(* PLC project Unnamed, Unknown Unnamed 1 *)
(* stored: creationDateTime 2023-03-10T10:37:17, modificationDateTime 2023-03-15T15:56:42 *)

(* 978-3-658-16137-8, Aufgabe 2.41 *)
FUNCTION_BLOCK Dice_Numbers_Indicator
  VAR_INPUT
    IN1 : BOOL;
    IN2 : BOOL;
    IN3 : BOOL;
    IN4 : BOOL;
  END_VAR
  VAR_OUTPUT
    OUTa : BOOL;
    OUTb : BOOL;
    OUTc : BOOL;
    OUTd : BOOL;
    OUTe : BOOL;
    OUTf : BOOL;
    OUTg : BOOL;
    OUTh : BOOL;
    OUTi : BOOL;
  END_VAR
  VAR  (* added by the conversion: wires and edge detectors of the diagram *)
    _OR40_OUT : BOOL;
    _OR53_OUT : BOOL;
    _OR70_OUT : BOOL;
  END_VAR

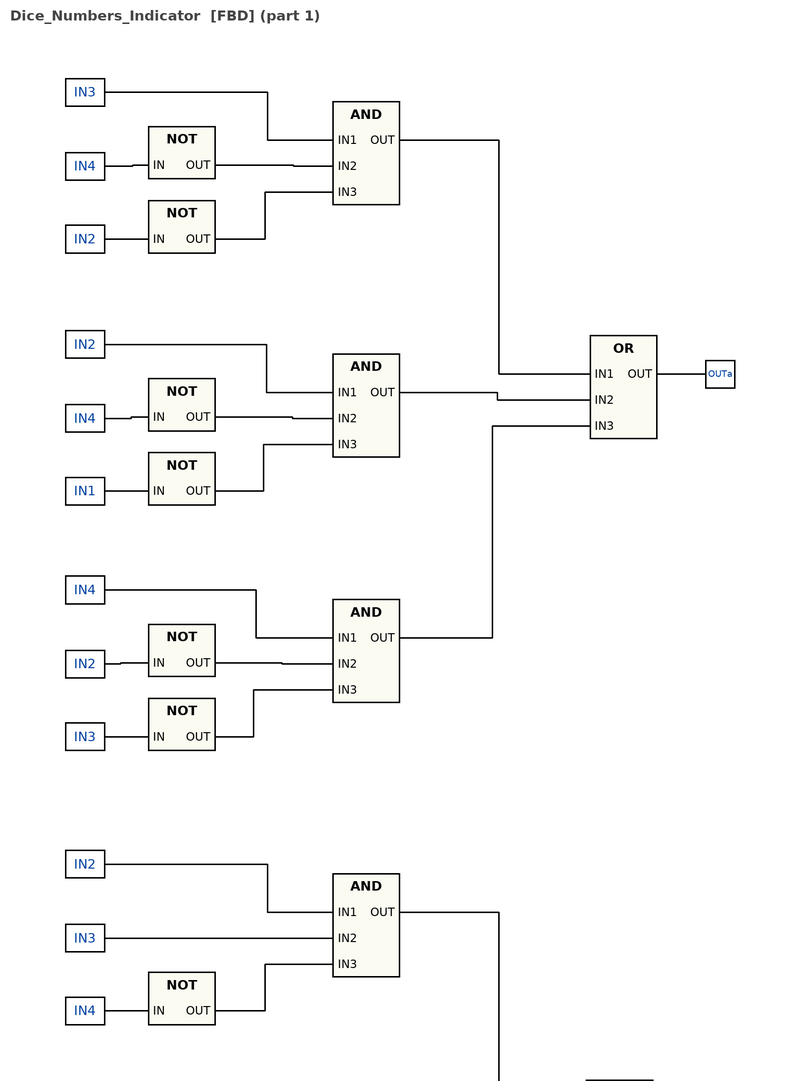
(* FBD diagram, written out as Structured Text *)
OUTa := IN3 AND NOT IN4 AND NOT IN2 OR IN2 AND NOT IN4 AND NOT IN1 OR IN4 AND NOT IN2 AND NOT IN3;
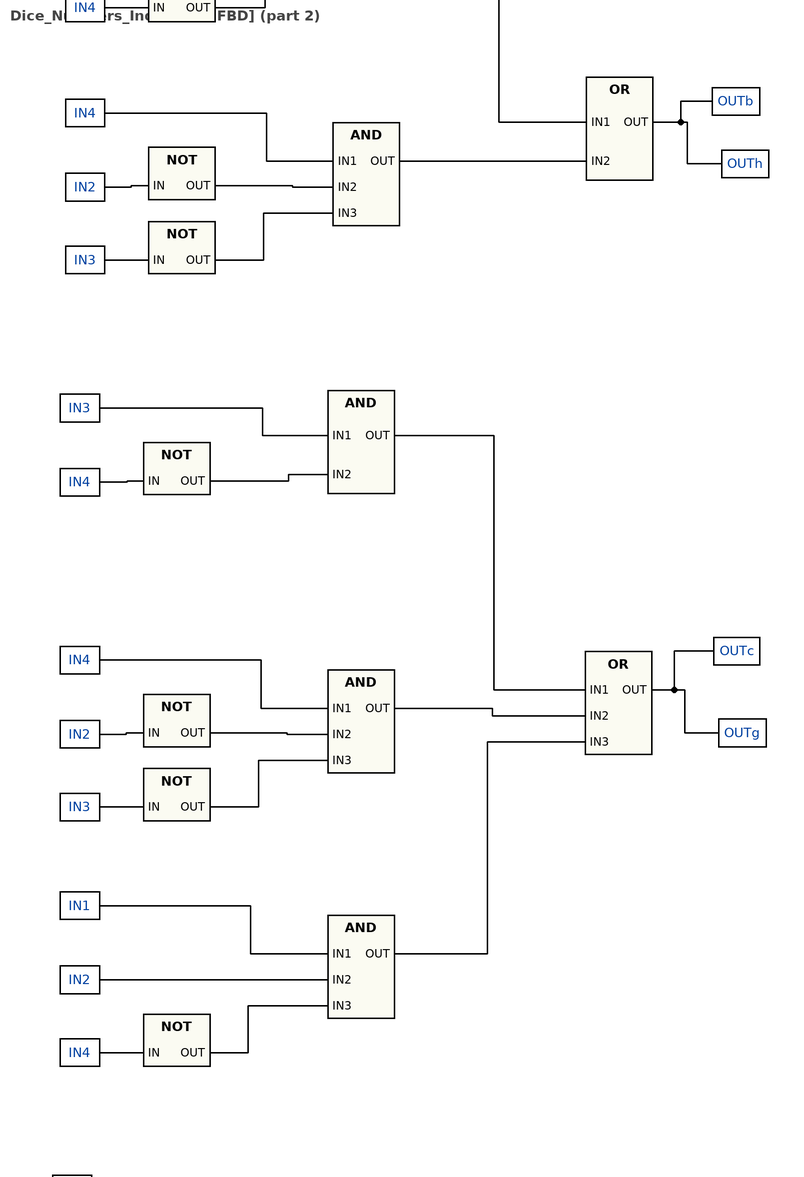
_OR40_OUT := IN2 AND IN3 AND NOT IN4 OR IN4 AND NOT IN2 AND NOT IN3;
OUTb := _OR40_OUT;
OUTh := _OR40_OUT;
_OR53_OUT := IN3 AND NOT IN4 OR IN4 AND NOT IN2 AND NOT IN3 OR IN1 AND IN2 AND NOT IN4;
OUTc := _OR53_OUT;
OUTg := _OR53_OUT;
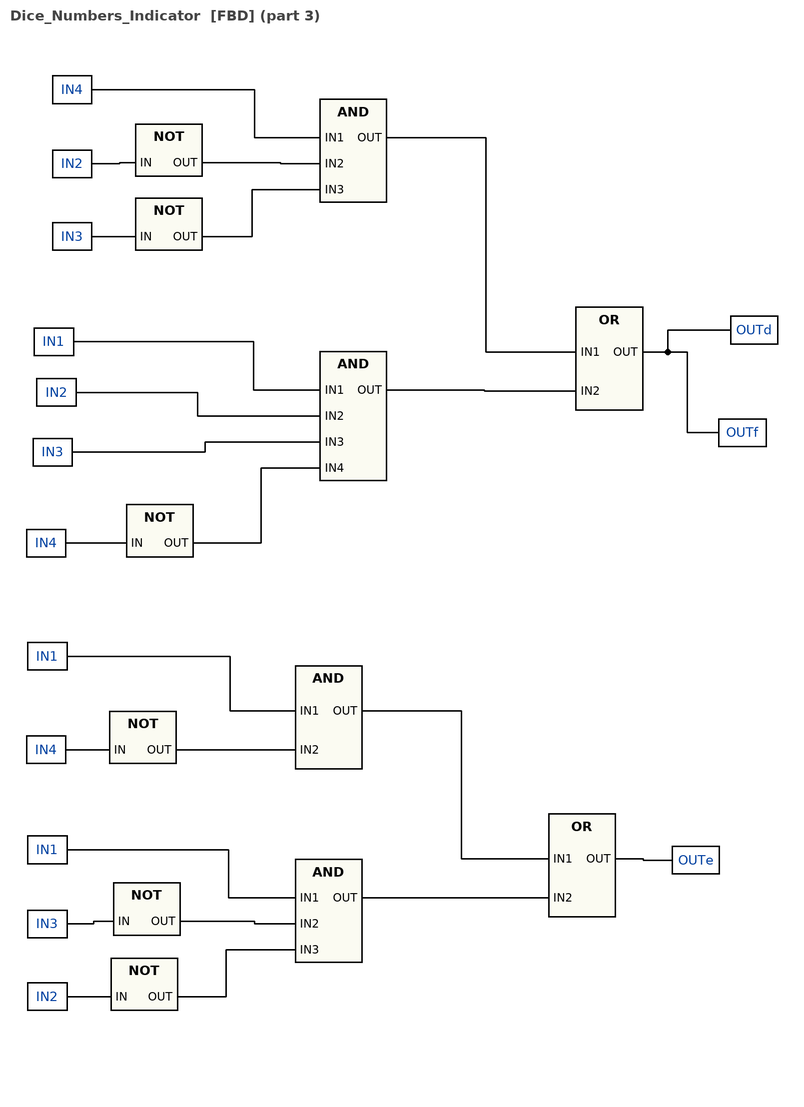
_OR70_OUT := IN4 AND NOT IN2 AND NOT IN3 OR IN1 AND IN2 AND IN3 AND NOT IN4;
OUTd := _OR70_OUT;
OUTf := _OR70_OUT;
OUTe := IN1 AND NOT IN4 OR IN1 AND NOT IN3 AND NOT IN2;
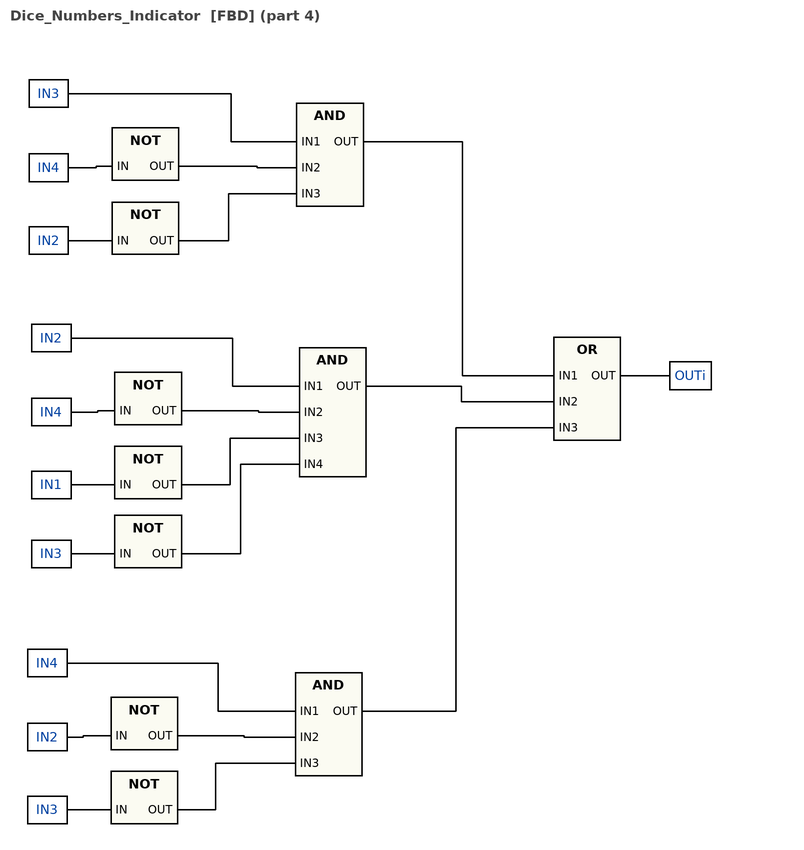
OUTi := IN3 AND NOT IN4 AND NOT IN2 OR IN2 AND NOT IN4 AND NOT IN1 AND NOT IN3 OR IN4 AND NOT IN2 AND NOT IN3;
END_FUNCTION_BLOCK

CONFIGURATION config
  RESOURCE resource1 ON PLC
  END_RESOURCE
END_CONFIGURATION
